PROGRAM Axis05_Status
VAR
	Always_ON	:	BOOL	:=TRUE	;//상시 ON 
	Always_OFF	:	BOOL	:=FALSE	;//상시 OFF
END_VAR

// NETWORK 1

END_PROGRAM

(* stored: Version 1.1.0.1, ProductVersion 3.1.4024.15
   POU Axis05_Status: Id {cfc680cf-dda7-423e-9182-aaaf7d5606b2}, SpecialFunc None *)
